// TwinCAT 3 PLC project PLC
// ProgramVersion: 3.1.4024.0
// libraries:
//   Tc2_MC2, * (Beckhoff Automation GmbH)
//   Tc2_Standard, * (Beckhoff Automation GmbH)
//   Tc2_System, * (Beckhoff Automation GmbH)
//   Tc3_Module, * (Beckhoff Automation GmbH)
// project tree:
//   GVLs/ Eixos.TcGVL
//   / PlcTask.TcTTO
//   POUs/ MAIN.TcPOU
// real-time tasks:
//   TASK PlcTask: cycle T#10ms, priority 20, ADS port 350
// motion (NC):
//   TASK NCTask SAF: cycle T#2ms, priority 4, ADS port 501
//   TASK NCTask SVB: cycle T#10ms, priority 8, ADS port 511
//   AXIS Eixo1 (id 1)
//   AXIS Eixo2 (id 2)
// variable links:
//   PLC Instance <-> NCTask SAF/Axes/Eixo1
//     PlcTask Inputs/Eixos.Eixo1.NcToPlc <-> Outputs/ToPlc
//     PlcTask Outputs/Eixos.Eixo1.PlcToNc <-> Inputs/FromPlc
//   PLC Instance <-> NCTask SAF/Axes/Eixo2
//     PlcTask Inputs/Eixos.Eixo2.NcToPlc <-> Outputs/ToPlc
//     PlcTask Outputs/Eixos.Eixo2.PlcToNc <-> Inputs/FromPlc

CONFIGURATION PLC
    RESOURCE PLC ON TwinCAT3
        TASK PlcTask(INTERVAL := T#10ms, PRIORITY := 20);
        PROGRAM MAIN WITH PlcTask : MAIN;
    END_RESOURCE
END_CONFIGURATION

// ---- GVLs/Eixos.TcGVL
VAR_GLOBAL
	Eixo1 : AXIS_REF;
	Eixo2 : AXIS_REF;
END_VAR

// ---- POUs/MAIN.TcPOU
PROGRAM MAIN
VAR
	MaquinaLigada: BOOL;
	bHabilita: BOOL;
	fb_Habilita1: MC_Power;
END_VAR

//Ler Status
	Eixos.Eixo1.ReadStatus();
	Eixos.Eixo2.ReadStatus();
	
//Habilitar Eixo1
IF MaquinaLigada THEN
		bHabilita := 1;
	ELSE
		bHabilita := 0;
	END_IF
	fb_Habilita1(
		Axis:= Eixos.Eixo1, 
		Enable:= bHabilita, 
		Enable_Positive:= bHabilita, 
		Enable_Negative:= bHabilita, 
		Override:= 100.0);

END_PROGRAM
